FUNCTION FC_GetLocalTimeString : T_SHORT_STR		// Returns the local time as string, eg. '15:58:40:302'

FC_GetLocalTimeString := IING.localTimeString;

END_FUNCTION

(* stored: Version 1.1.0.1, ProductVersion 3.1.4026.18
   POU FC_GetLocalTimeString: Id {84e9b491-40f4-4f5e-990c-98f9bf29b462}, SpecialFunc None *)
